// TIA Portal V20 export
TYPE "LKinCtrl_typeToolParameters"
   STRUCT
      offsetParaNo : Int;   // selection of offset parameter set from configuration structure
      mainPathPlane : Int;   // main path plane for compensation
   END_STRUCT;
END_TYPE
